(* IEC 61131-3 sources: iec-st-tools/testdata/src/UserGlobals, 1 file *)

(* ---- Globals.st ---- *)
CONFIGURATION Globals
    VAR_GLOBAL
        G_SafeInvertTest : INT := 0;
    END_VAR
END_CONFIGURATION
